(* IEC 61131-3 sources: SJ_AGV/PLC/Standard_functions.4.4.0/Common, 6 files *)

(* ---- DEBUG_FB.ST ---- *)
FUNCTION_BLOCK DEBUG_FB
VAR_EXTERNAL

END_VAR

VAR_INPUT

END_VAR

VAR_OUTPUT

END_VAR

VAR

END_VAR
if debug then
	a:= TRACE_bool('ExecDrvCmd',NDC8.Automatic.ExecDriveCommand);
	a:= TRACE_bool('CancOp',NDC8.LoadOperation.CancelOperation);
	a:= TRACE_dint('TrvlDir',NDC8.VehicleControl.TravelDir);
	a:= TRACE_BOOL('Loaded', input.LoadOnBoard);
	a:= TRACE_DINT('Segm', NDC8.LayoutPosition.Segment);
	a:= TRACE_BOOL('OnLastseg', NDC8.LoadDocking.OnLastSegment);
	a:= TRACE_DINT('StopWord', NDC8.UserDefined.StopWord);
	a:= TRACE_DINT('OpCode', NDC8.LoadOperation.OperationCode);
	a:= TRACE_DINT('OpPar1', NDC8.LoadOperation.OperationParam1);

	debug := false;

end_if;

END_FUNCTION_BLOCK

(* ---- INDICATORS_FB.ST ---- *)
FUNCTION_BLOCK INDICATORS_FB
VAR_EXTERNAL
	(** IN **)
	NDC8 : NDC8_T;
	INPUT : INPUT_T;
	Output : OUTPUT_T;

END_VAR

VAR_INPUT
	SetHeight						: dint;
	ForkTarget,
	AutoInsertNotInsideTargetSafety,
	AutoinsertInProgress,
	SensorsBuzzerTest,
	StartDelayStartWarning,
	LS2000SlowDown					: bool;

END_VAR

VAR_OUTPUT

END_VAR

VAR
	FlashError,
	FlashWarning,
	FlashRight,
	FlashLeft,
	FlashForward,
	FlashBackward,
	FlashSegment : Bool;
	FlashBrakeRel : BOOL;
	ModeAutoTON :TON;

	Display : bool;
	SlowBeep : bool;

END_VAR
(*
------------------------------------------------------------------------------------
 INDICATORS_FB
 ------------------

 Description:
 This PLC controls the flashing of the lights and the sounding of the buzzer.
 The lights and buzzer functionality is made according to safety regulations EN-1525.

-------------------------------------------------------------------------------------*)

(* make default *)
Output.PositionKnownLamp 	:= false;
Output.EmergencyStopLamp 	:= false;
Output.LoadOnBoardLamp	 	:= false;
Output.InSystemLamp			:= false;
Output.FrontLeftLamp 		:= false;
Output.FrontRightLamp 		:= false;
Output.RearLeftLamp 		:= false;
Output.RearRightLamp 		:= false;
Output.WarningBuzzerTop		:= false;
Output.WarningLightTop		:= false;
Output.Buzzer 				:= false;
Output.OPTBuzzer			:= false;

(***************************************************************************************
	Evaluate which signals to set
****************************************************************************************)
(*Emergency stop or any stop flags*)
FlashError	:=	NDC8.VehicleControl.Estop
				or StopRear
				or StopSide
				or StopObstacle
				or StopLift
				or StopLoadChange
				or StopReset
				or StopSteerSync
				or StopForkFarTooHigh
				or StopForkTooHigh
				or StopForkTooLow
				or NDC8.Opt.VehicleStatusID = 11;

FlashBrakeRel := INPUT.Auto = TRUE and NDC8.SDIO.DigitalInput5_BTN_BRK = TRUE;

(*Segment trigger flash*)
FlashSegment := NDC8.VehicleControl.Moving;

(*Segment trigger or Vehical right turn*)
FlashRight 	:= 	Input.SD_Right or Input.DD_Right;

(*Segment trigger or Vehical right turn*)
FlashLeft 	:=	Input.SD_Left or Input.DD_Left;

(*Segment trigger or Vehical Forward*)
FlashForward := Input.SD_Forward;

(*Segment trigger or Vehical Backward*)
FlashBackward := Input.SD_Backward;

(* Special case for when we want to flash both right _and_left *)
(*If FlashRight and FlashLeft then
	  FlashRight	:= NDC8.TurnSignal.RightTurnDistance < NDC8.TurnSignal.LeftTurnDistance;
	  FlashLeft		:= NDC8.TurnSignal.LeftTurnDistance < NDC8.TurnSignal.RightTurnDistance;
End_if;*)

(*Vehicle moving backwards, forks are moving or before starting to drive *)
FlashWarning := (SetHeight > 0 and not ForkTarget )
				or (NDC8.VehicleControl.Moving and NDC8.VehicleControl.TravelDir = 0)
				or INPUT.SafetyScannerSlowDown
				or StartDelayStartWarning
				or (NDC8.Guidance.StopReason = 1
  					and NDC8.Guidance.DistanceToStop < 1500
  					and NDC8.VehicleControl.TravelDir = 1);		(* Vehicle will stop and change travel directions and reverse. *)

(***************************************************************************************)
(*			LAMPS 					*)
(***************************************************************************************)
(* GREEN lamp;	Position known *)
if 	NDC8.Position.Valid then
	if NDC8.VehicleControl.OperationMode = 0 then
		Output.PositionKnownLamp := true;										(* Automatic mode: 		ON 		*)
	else
	 	Output.PositionKnownLamp := Timer.Info;								(* Semi/manual mode: 	BLINK 	*)
	end_if;
end_if;

(***************************************************************************************)
(* WHITE lamp; reset button *)

Output.ResetButtonLamp	:= (StopReset or												(* need reset	*)
					   		StopManual or
					   		AutoInsertNotInsideTargetSafety 								(* vehicle need assistance during autoinsert *)
							)
							and Timer.Info;

(***************************************************************************************)
(* YELLOW lamp; Load on board*)
Output.LoadOnBoardLamp := INPUT.LoadOnBoard and Timer.Info;

(***************************************************************************************)
(* RED lamp; S100 stop *)
Output.EmergencyStopLamp := NDC8.VehicleControl.OperationMode = 0 and StopObstacle and Timer.Error;								(* S100 stop *)

(***************************************************************************************)
(* BLUE lamp; In system *)

if NDC8.VehicleControl.OperationMode = 0 then
	Output.InSystemLamp :=	NDC8.LayoutPosition.InSystem 							(* in system *)
				or (AutoinsertInProgress and NDC8.VehicleControl.Moving and Timer.Warning)

				or (INPUT.Reset_PB  								(*	 on when pressed and outside safety	*)
					and AutoInsertNotInsideTargetSafety
					)
				or (AutoinsertInProgress				(* 	 need more RESET help 	*)
					and not NDC8.VehicleControl.Moving
					and Timer.Info);
end_if;

(***************************************************************************************)
(* SIDE ORANGE lamp; warning/turn indicators *)
InStatus := NDC8.VehicleControl.OperationMode = 0;
ModeAutoTON(IN:=InStatus,PT:=t#2s);	(* Wait 2 sec before flashing when entering auto*)
if TRUE then
	if FlashError then
		Output.RearLeftLamp 	:= Timer.Error;
		Output.RearRightLamp	:= Timer.Error;
		Output.FrontLeftLamp 	:= Timer.Error;
		Output.FrontRightLamp	:= Timer.Error;
		(* vehicle moving or vehicle error both flash *)
		(*
	elsif FlashWarning or FlashSegment then
		Output.RearLeftLamp 	:= Timer.Warning;
		Output.RearRightLamp	:= Timer.Warning;
		Output.FrontLeftLamp 	:= Timer.Warning;
		Output.FrontRightLamp	:= Timer.Warning;*)
	elsif FlashBrakeRel then
		Output.FrontLeftLamp 	:= TRUE;
		Output.RearLeftLamp 	:= TRUE;
		Output.FrontRightLamp 	:= TRUE;
		Output.RearRightLamp 	:= TRUE;
	elsif FlashForward then								(* vehicle turning to the left *)
		Output.FrontLeftLamp 	:= Timer.Warning;
		Output.RearLeftLamp 	:= Timer.Warning;
		Output.FrontRightLamp 	:= Timer.Warning;
		Output.RearRightLamp 	:= Timer.Warning;
	elsif FlashBackward then								(* vehicle turning to the left *)
		Output.FrontLeftLamp 	:= Timer.Warning;
		Output.RearLeftLamp 	:= Timer.Warning;
		Output.FrontRightLamp 	:= Timer.Warning;
		Output.RearRightLamp 	:= Timer.Warning;
	elsif FlashRight then								(* vehicle turning to the right *)
		Output.FrontLeftLamp 	:= false;
		Output.RearLeftLamp 	:= false;
		Output.FrontRightLamp 	:= Timer.Warning;
		Output.RearRightLamp 	:= Timer.Warning;
	elsif FlashLeft then								(* vehicle turning to the left *)
		Output.FrontLeftLamp 	:= Timer.Warning;
		Output.RearLeftLamp 	:= Timer.Warning;
		Output.FrontRightLamp 	:= false;
		Output.RearRightLamp 	:= false;
	elsif NDC8.VehicleControl.Moving = FALSE then
		Output.FrontLeftLamp 	:= TRUE;
		Output.RearLeftLamp 	:= TRUE;
		Output.FrontRightLamp 	:= TRUE;
		Output.RearRightLamp 	:= TRUE;
	end_if;
elsif StopReset then									(* Reset required *)
		Output.FrontLeftLamp 	:= Timer.Info and Timer.Error and Timer.Warning;
		Output.FrontRightLamp 	:= Timer.Info and Timer.Error and Timer.Warning;
		Output.RearLeftLamp 	:= Timer.Info and Timer.Error and Timer.Warning;
		Output.RearRightLamp 	:= Timer.Info and Timer.Error and Timer.Warning;
end_if;

if StopLS2000 or LS2000SlowDown then							(* Vehicle is about to drive into something and hit LS2000! *)
		Output.RearLeftLamp 	:= Timer.Warning;
		Output.RearRightLamp	:= Timer.Warning;
		Output.FrontLeftLamp 	:= Timer.Warning;
		Output.FrontRightLamp	:= Timer.Warning;
end_if;

(***************************************************************************************)
(* 					BUZZERS 					*)
(***************************************************************************************)
(* High frequency tone. Sound only when there is a drive command. *)
InStatus := NDC8.VehicleControl.OperationMode = 0;
ModeAutoTON(IN:=InStatus,PT:=t#3s);	(* Wait 3 sec before buzzing when entering auto *)
Output.Buzzer	:=	(ModeAutoTON.Q and
						NDC8.Automatic.ExecDriveCommand	and
							(FlashError and Timer.Error)				(* Error *)
						 	or
						 	(FlashWarning and Timer.Warning)					(* Info *)
						)
					or SensorsBuzzerTest
					or (StopLS2000 or LS2000SlowDown and Timer.Warning);			(* Vehicle is about to drive into something and hit LS2000! *)

(* OPT 100 BUZZER Low frequency tone *)
OUTPUT.OPTBuzzer	:= StartDelayStartWarning					(* Sound during start or if reset is required. *)
						or
							(StopReset or StopLS2000 or LS2000SlowDown)
							and Timer.Info
							and Timer.Error
							and Timer.Warning
							and SlowBeep;

END_FUNCTION_BLOCK

(* ---- MODECONTROL_FB.ST ---- *)
FUNCTION_BLOCK MODECONTROL_FB
VAR_EXTERNAL
	NDC8 : NDC8_T;
	INPUT : INPUT_T;
	TRUCK : TRUCK_T;

END_VAR

VAR_INPUT

END_VAR

VAR_OUTPUT
		Auto			: bool; (* 8 *)
		Manual			: bool; (* 1 *)
		Semi			: bool; (* 2 *)
		PPA				: bool; (* 4 *)

END_VAR

VAR
	State			: dint;
	SteerModeRT		: r_trig;
	SteerModeRT2	: r_trig;
	SteerMode	: dint;

	StepDelay : TON;

	NoMcdTimer : TON;

END_VAR
(*****************************************************************************************)
(* Truck Modes of Operation:

	Auto  					- full AGV control
	Manual					- Vehicle driven from tiller arm or MCD.
	PPA Tune  				- AGV drive mode, but vehicle controller set to manual mode to allow PPA Tuning

	NDC8.Manual.PlcSelectMask	DINT 	Individually select mask:
		Bit0:PlcAngle 				2#00000
		Bit1:PlcSpeed 				2#00010
		Bit2:PlcSetOperationMode 	2#00100
		Bit3:Reserved 				2#01000
		Bit4:PlcSteerMethod			2#10000
	*)

NDC8.Manual.PlcSelect := true;							(* By default, allow overrides.*)
NDC8.Manual.PlcSelectMask := 0;							(* By default, don't override anything*)

(* only one mode is allowed at one time *)
Auto 			:= word_to_bool(dint_to_word(State) and 16#8);
Manual			:= word_to_bool(dint_to_word(State) and 16#1);
Semi			:= word_to_bool(dint_to_word(State) and 16#2);
PPA 			:= word_to_bool(dint_to_word(State) and 16#4);

INPUT.Auto := Auto;
INPUT.Manual := Manual;
INPUT.Semi := Semi;
INPUT.PPA := PPA;

if NDC8.Mcd.Valid = TRUE and g_StartFindSync = FALSE then

	SteerModeRT(CLK:=Input.ChangeSteerMode_PB);		(* New steer mode requested (Quad vehicle)
															0: 2*SD Anti-parallel
															1: 2*SD Parallel
															2: DiffDrive  				*)
	SteerModeRT2(CLK:=Input.ChangeSteerMode_PB2);

	case State of
	(*****************************************************************************************
				Automatic mode
	*****************************************************************************************)
	0: State := 8;

	8:	NDC8.Manual.PlcSetOperationMode := 0;			(* Operation mode Auto *)
		NDC8.Manual.PlcSelectMask		:= 2#00110;	(* Override Set speed, to allow autinsert from outside safety zone
														 Speed is set in AutoInsert FB. *)

		(**** Exit this mode? ***)
		if NDC8.Mcd.Button2 and NDC8.Mcd.Valid then		(* MCD semi mode *)
			State := 2;

		elsif (NDC8.Mcd.Button3 and NDC8.Mcd.Valid)		(* MCD manual mode *)
			or INPUT.TillerArmDown 						(* Manual arm down, switch to manual mode		*)
			or INPUT.GateOpen
			or INPUT.PlatformNotUpperPos then
				State := 1;

		elsif NDC8.Userdefined.PPAEnable = 2 then		(* Change to PPA mode if set in OPT	expert menu.*)
				State := 4;
		end_if;

	(*****************************************************************************************
				Semi mode (MCD throttle, automatic steering)
	*****************************************************************************************)
	2:	NDC8.Manual.PlcSetOperationMode := 2;			(* Set semi mode *)
		NDC8.Manual.PlcSelectMask 		:= 2#10010;	(* Override operation mode and steer mode (quad) *)

		(**** Exit this mode? ***)
		if NDC8.Mcd.Button1 or not NDC8.Mcd.Valid then		(* If disconnect the MCD or switch modes, to auto *)
			State := 8;

		elsif (NDC8.Mcd.Button3 and NDC8.Mcd.Valid) then	(* If disconnect the MCD or switch modes, to auto *)
			State := 1;
		end_if;

	(*****************************************************************************************
				Manual driving
	*****************************************************************************************)
	1:	NDC8.Manual.PlcSetOperationMode := 1;				(* Set Manual mode 							*)
		StopLoadOP := False;								(* Clear load op cancel stop bit			*)

		if SteerModeRT.q then
			SteerMode:= SteerMode + 1;          			(* Toggle steermode *)
	        if SteerMode > 2 then                  			(* Limit *)
	        	SteerMode:= 0;                				(* Reset *)
			end_if;
	        NDC8.Manual.PLCSteerMode:= SteerMode;   		(* Use steermode *)
		end_if;

		if SteerModeRT2.q then
			SteerMode:= SteerMode - 1;          		(* Toggle steermode *)
	        if SteerMode < 0 then                  		(* Limit *)
	        	SteerMode:= 2;                			(* Reset *)
			end_if;
	        NDC8.Manual.PLCSteerMode:= SteerMode;   	(* Use steermode *)
		end_if;

		if NDC8.Mcd.Valid then								(* If mcd connected						 	*)
			if Input.ZeroSteerAngle_PB then					(* If "set zero angle" key					*)
				NDC8.Manual.PLCAngle 			:= 0;		(* Set angle to 0							*)

				if StopWord = 0 and StopWord2 = 0  then
					NDC8.Manual.PlcSpeed			:= NDC8.Mcd.Speed;
				elsif NDC8.Mcd.Button8 = FALSE then
					NDC8.Manual.PlcSpeed			:= 0;
				elsif NDC8.Mcd.Button8 = TRUE then
					NDC8.Manual.PlcSpeed			:= NDC8.Mcd.Speed;
				end_if;

				NDC8.Manual.PlcSelectMask 		:= 2#10111;(* Override operation mode, steer mode and set angle	*)
			else
				NDC8.Manual.PLCAngle 			:= NDC8.Mcd.Angle / 3;

				if StopWord = 0 and StopWord2 = 0  then
					NDC8.Manual.PlcSpeed			:= NDC8.Mcd.Speed;
				elsif NDC8.Mcd.Button8 = FALSE then
					NDC8.Manual.PlcSpeed			:= 0;
				elsif NDC8.Mcd.Button8 = TRUE then
					NDC8.Manual.PlcSpeed			:= NDC8.Mcd.Speed;
				end_if;

				NDC8.Manual.PlcSelectMask 		:= 2#10111;(* Override operation mode and steer mode		*)
			end_if;
			DisplayStopString(INStatus:=Input.ZeroSteerAngle_PB, StopString:=184, StopValue:=0);
			StopManual := false;

		else
			NDC8.Manual.PlcSelectMask 		:= 2#10101;			(* Override operation mode, set angle and steer mode		*)
			NDC8.Manual.PlcAngle := Input.SteerEncAngle;		(* Follow encoder angle, to start autoinsert with this set angle. *)

			StopManual	:= not Input.GateOpen 					(* Set stop bit while waiting to go to auto.	*)
						and not Input.TillerArmDown
						and not Input.PlatformNotUpperPos
						and not Input.Reset_PB;
			StopReset	:= StopReset OR StopManual; 			(* This stop signal needs to be reset			*)
		end_if;

		(**** Exit this mode? ***)
		if NDC8.Mcd.Valid then									(* If MCD is connected							*)
			if NDC8.Mcd.Button1 then							(* Auto mode on MCD? Switch to automatic mode.	*)
				State := 8;
			elsif NDC8.Mcd.Button2 then							(* Semi mode on mcd? Switch to semi mode		*)
				State := 2;
			end_if;
		else
			if 	not Input.TillerArmDown							(* Tiller arm up								*)
				and not Input.GateOpen							(* and gate closed 								*)
				and not Input.PlatformNotUpperPos				(* and platform up 								*)
				and Input.Reset_PB then							(* and reset push button! 						*)
					State := 8;							(* Switch to automatic mode						*)
			end_if;
		end_if;

	(*****************************************************************************************
				Physical Parameter Adjust (PPA)
	*****************************************************************************************)

	4:	NDC8.Manual.PlcSetOperationMode  := 1;			(* Set Manual mode								*)
		NDC8.Manual.PlcSelectMask 		 := 2#00100;	(* Override operation mode 						*)

		(**** Exit this mode? ***)
		if INPUT.TillerArmDown
			or INPUT.GateOpen
			or INPUT.PlatformNotUpperPos then
				State := 1;						(* Manual arm down, switch to manual mode		*)

		elsif NDC8.Userdefined.PPAEnable <> 2 then		(* PPA symbol changed? Go back to auto.			*)
				State := 8;
		end_if;

	end_case;

	NoMcdTimer(IN:= FALSE);
elsif NDC8.Mcd.Valid = FALSE and g_StartFindSync = FALSE and g_ErrorCode = 0 then

	NoMcdTimer(IN:= TRUE, PT:=t#5s);

;
end_if;

(**************************************************************************************)
(* Update Display *)

DisplayStopString(INStatus:=StopManual, StopString:=85, StopValue:=0);

END_FUNCTION_BLOCK

(* ---- STOPWORD_FB.ST ---- *)
FUNCTION_BLOCK STOPWORD_FB
VAR_EXTERNAL
	NDC8 : NDC8_T;
END_VAR

VAR_INPUT
END_VAR

VAR_OUTPUT
END_VAR

VAR
	WaitingForSteerWheelTurn : bool;
	Stop_RT : R_Trig;
	Stop_FT : F_Trig;
	TempValue : dint ;
	StopTON : ton;
END_VAR
(**************************************************************************************)
(* LOAD OPERATION STOP *)
(* Do not enter station w/o OP code *)
(*StopNoOPCode := NDC8.LoadOperation.OperationCode = 0
				and NDC8.Automatic.ExecDriveCommand;
DisplayStopString(InStatus:=StopNoOPCode, StopString:=94, StopValue:=0);

*)

(**************************************************************************************)
(* Waiting for steering wheel to turn *)
(* If no other errors, it's most likely the steer wheel which is not within NDC8.Vehicle.WaitForWheelTurnMaxAngle. *)

WaitingForSteerWheelTurn := NDC8.Automatic.ExecDriveCommand
							and NDC8.CanOpenMaster.NMTState = 5
							and NDC8.CanOpenMaster.State = 0
							and NDC8.Position.Valid
							and not NDC8.Vehicle.Blocked
							and not NDC8.VehicleControl.QuickStop
							and not NDC8.VehicleControl.Stop
							and not NDC8.VehicleControl.EStop
							and not NDC8.VehicleControl.SensorStopEnable
							and NDC8.VehicleControl.SetSpeed = 0
							and abs(Input.SteerEncAngle - Output.SetValueSteer) > NDC8.Vehicle.WaitForWheelTurnMaxAngle;

DisplayStopString(InStatus:=WaitingForSteerWheelTurn, StopString:=138, StopValue:=0);

StopSteerSync	:= not INPUT.SteerEncSyncValid;
DisplayStopString(InStatus:=StopSteerSync, StopString:=181, StopValue:=0);

DisplayStopString(InStatus:=StopByOM_PLC, StopString:=200, StopValue:=0);
DisplayStopString(InStatus:=StopByErrorCode, StopString:=201, StopValue:=0);
DisplayStopString(InStatus:=StopBatLowOT, StopString:=202, StopValue:=0);
DisplayStopString(InStatus:=StopFindSync, StopString:=203, StopValue:=0);
DisplayStopString(InStatus:=StopRobotNotIdle, StopString:=204, StopValue:=0);
DisplayStopString(InStatus:=StopByBCD, StopString:=205, StopValue:=0);

DisplayStopString(InStatus:=StopLift, 				StopString:=210, StopValue:=0);
DisplayStopString(InStatus:=StopRear,				StopString:=211, StopValue:=0);
DisplayStopString(InStatus:=StopSafety, 			StopString:=212, StopValue:=0);
DisplayStopString(InStatus:=StopFailureCAN, 		StopString:=213, StopValue:=0);
DisplayStopString(InStatus:=StopStartDelay,	 		StopString:=214, StopValue:=0);
DisplayStopString(InStatus:=StopFlex, 				StopString:=215, StopValue:=0);
DisplayStopString(InStatus:=StopSoft, 				StopString:=216, StopValue:=0);
DisplayStopString(InStatus:=StopLoadChange,	 		StopString:=217, StopValue:=0);
DisplayStopString(InStatus:=StopObstacle, 			StopString:=218, StopValue:=0);
DisplayStopString(InStatus:=StopEStopChainError, 	StopString:=219, StopValue:=0);
DisplayStopString(InStatus:=StopSteerSync, 			StopString:=220, StopValue:=0);
DisplayStopString(InStatus:=StopEstopButton, 		StopString:=221, StopValue:=0);
DisplayStopString(InStatus:=StopSide, 				StopString:=222, StopValue:=0);
DisplayStopString(InStatus:=StopReset,				StopString:=223, StopValue:=0);
DisplayStopString(InStatus:=StopNoOpCode, 			StopString:=224, StopValue:=0);
DisplayStopString(InStatus:=StopManual, 			StopString:=225, StopValue:=0);
DisplayStopString(InStatus:=StopCharge, 			StopString:=226, StopValue:=0);
DisplayStopString(InStatus:=StopClamp, 				StopString:=227, StopValue:=0);
DisplayStopString(InStatus:=StopFailCode, 			StopString:=228, StopValue:=0);
DisplayStopString(InStatus:=StopResetButton, 		StopString:=229, StopValue:=0);
DisplayStopString(InStatus:=StopLoadOP, 			StopString:=230, StopValue:=0);
DisplayStopString(InStatus:=StopBumperFault, 		StopString:=231, StopValue:=0);
DisplayStopString(InStatus:=StopObstacleFault, 		StopString:=232, StopValue:=0);
DisplayStopString(InStatus:=StopTruckDriveSafeState,StopString:=233, StopValue:=0);
DisplayStopString(InStatus:=StopLS2000, 			StopString:=234, StopValue:=0);
DisplayStopString(InStatus:=StopHalt, 				StopString:=235, StopValue:=0);
DisplayStopString(InStatus:=StopLoadDroppedWhileUnloading, StopString:=236, StopValue:=0);
DisplayStopString(InStatus:=StopSpinningWheel, 		StopString:=237, StopValue:=0);
DisplayStopString(InStatus:=StopForkTooLow, 		StopString:=238, StopValue:=0);
DisplayStopString(InStatus:=StopForkTooHigh, 		StopString:=239, StopValue:=0);
DisplayStopString(InStatus:=StopForkFarTooHigh, 	StopString:=240, StopValue:=0);
DisplayStopString(InStatus:=StopChargeStationMissing, StopString:=241, StopValue:=0);

DisplayStopString(InStatus:=StopByCanErr_Node1, StopString:=244, StopValue:=0);
DisplayStopString(InStatus:=StopByCanErr_Node2, StopString:=245, StopValue:=0);
DisplayStopString(InStatus:=StopByCanErr_Node3, StopString:=246, StopValue:=0);
DisplayStopString(InStatus:=StopByCanErr_Node4, StopString:=247, StopValue:=0);
DisplayStopString(InStatus:=StopByCanErr_Node5, StopString:=248, StopValue:=0);
DisplayStopString(InStatus:=StopByCanErr_Node6, StopString:=249, StopValue:=0);
DisplayStopString(InStatus:=StopByCanErr_Node7, StopString:=250, StopValue:=0);
DisplayStopString(InStatus:=StopByCanErr_Node8, StopString:=251, StopValue:=0);
DisplayStopString(InStatus:=StopByCanErr_Node9, StopString:=252, StopValue:=0);
DisplayStopString(InStatus:=StopByCanErr_Node10, StopString:=253, StopValue:=0);

(**************************************************************************************)
(* QUICK STOP  (Stop with emergency deceleration ramp) 								  *)
(*NDC8.VehicleControl.QuickStop := StopFlex or StopObstacle or StopSafety;
*)
DisplayStopString(INStatus:=NDC8.VehicleControl.QuickStop, StopString:=179, StopValue:=0);

(**************************************************************************************)
(* STOP WORD sets stop signal 														  *)
NDC8.VehicleControl.Stop 	:= 	(Input.Auto and (DWORD_TO_BOOL(StopWord) or DWORD_TO_BOOL(StopWord2))) or
								(Input.Manual and NDC8.Mcd.Button8 = FALSE and (DWORD_TO_BOOL(StopWord) or DWORD_TO_BOOL(StopWord2)));
NDC8.UserDefined.StopWord	:=	DWORD_TO_DINT(StopWord);
NDC8.OMPLC.StopWord			:=	DWORD_TO_INT(StopWord);

StopTON(IN:=NDC8.VehicleControl.Stop,PT:=t#10s);
Stop_RT(CLK:=StopTON.q);
if Stop_RT.Q and not StopStartDelay then
	TempValue:=DWord_To_DINT(StopWord);
end_if;

(* Send event that stopword has been cleared. * )
Stop_FT(CLK:=NDC8.VehicleControl.Stop);
if Stop_FT.q then
	EventQueue(EventCode:=101,Par1:=NDC8.Vehicle.VehicleID,Par2:=0,Par3:=0,Par4:=0);
end_if;
*)

END_FUNCTION_BLOCK

(* ---- Timer_FB.ST ---- *)
FUNCTION_BLOCK Timer_FB
VAR_OUTPUT
	Error : bool;
	Warning : bool;
	Info : bool;
	Display : bool;
	SlowBeep : bool;

END_VAR

VAR
	TimerError 		: blink;
	TimerWarning 	: blink;
	TimerInfo 		: blink;
	TimerDisplay	: blink;
	TimerSlowBeep	: blink;
END_VAR
(*
------------------------------------------------------------------------------------
 FREERUN
 -------

 Description:
 Creates different outputs that will look like a freerunning timer.
 Outputs will toggle with different timebase.
 They are all defined globally.
------------------------------------------------------------------------------------   *)

TimerError	(CYCLE :=t#240ms,RUN:=true);
TimerWarning(CYCLE :=t#480ms,RUN:=true);
TimerInfo	(CYCLE :=t#960ms,RUN:=true);
TimerDisplay(CYCLE :=t#2s,RUN:=true);
TimerSlowBeep(CYCLE :=t#5s,RUN:=true);

Error		:= TimerError.Q1;
Warning	:= TimerWarning.Q1;
Info		:= TimerInfo.Q1;
Display	:= TimerDisplay.Q1;
SlowBeep	:= TimerSlowBeep.Q1;

END_FUNCTION_BLOCK

(* ---- TX_STATUS_FB.ST ---- *)
FUNCTION_BLOCK TX_STATUS_FB
VAR_EXTERNAL
	NDC8 : NDC8_T;
	Input : Input_T;

END_VAR

VAR_INPUT

END_VAR

VAR_OUTPUT

END_VAR

VAR

	Load_F : F_Trig;
	Load_F_FLAG : BOOL;

	Load_F_Timer : TON;

	BCD_Compare_R : F_Trig;
	BCD_Fail_R : F_Trig;

	BatLowR : R_Trig;
	BatLowF : F_Trig;

	ErrorCodeD : DINT;
	LastErrorCode : Word := 0;
	ErrorTrigFlag : bool;
	ErrorTrigR : R_Trig;
	ErrorTrigF : F_Trig;

	InsertDone : BOOL;
	InsertDoneR : R_Trig;

	PowerOffR	: R_Trig;

	WaitChargeR	: R_Trig;
	WaitChargeF	: F_Trig;

	ChargingR : R_Trig;
	ChargingF : F_Trig;

	ChargeDoneR : R_Trig;

	LoadStatusR :R_Trig;
	LoadStatusF :F_Trig;

	ManualModeR :R_Trig;
	ManualModeF :F_Trig;

	LostR :R_Trig;
	LostF :F_Trig;

	LocalModeR :R_Trig;
	LocalModeF :F_Trig;

	LocalInterlockFailCodeD : DINT;
	LocalInterlockFailFlag : bool;
	LocalInterlockFailR :R_Trig;

	DriveOutR : R_Trig;

	BrakeReleaseR : R_Trig;
	BrakeReleaseF : F_Trig;

	BeamStop_R : R_Trig;
	BeamStop_F : F_Trig;

	BlockFlagR : R_Trig;
	BlockFlagF : F_Trig;
	BlockModeFlag : BOOL;

	BCDReadFailR :R_Trig;

	(* Battery *)
	ChrgFlag_R_L : BOOL;
	TX_LowBatt_R : R_Trig;
	TX_ChgComp_R : R_Trig;
	Chrg_Right_Left_R : R_Trig;
	TX_Load_R : R_Trig;

	DINT_BMS2 : DINT;
	DINT_BMS3 : DINT;
	DINT_BMS_BatV : DINT;
	DINT_BMS_BatT : DINT;
	DINT_BMS_BatC : DINT;
	DINT_BMS_BatA : DINT;
	DINT_BMS_Main : DINT;
	DINT_BMS_Chan : DINT;
	DINT_BMS_ID4L : DINT;
	DINT_BMS_ID4H : DINT;

END_VAR
(*
------------------------------------------------------------------------------------
 TX_status
 ------------------

 Description:
 Sends status bits to master controller.

-------------------------------------------------------------------------------------*)
(*TxStatus bits*)

OM_PLC_Word1 := INT_TO_WORD(NDC8.OMPLC.ChargeOM);
OM_PLC_Word2 := INT_TO_WORD(NDC8.OMPLC.Stop_OM);

NDC8.PLC_Application.TxStatusBit0_Load := INPUT.LoadOnBoard;
NDC8.PLC_Application.TxStatusBit1_EaLD := PLC_RX01_Bit_EnableLD_i;

if NDC8.LoadOperation.OperationCode <> 0 then
	NDC8.PLC_Application.TxStatusBit2_HaveCmd := true;	(*Operation Code OK*)
else
	NDC8.PLC_Application.TxStatusBit2_HaveCmd := false;	(*Operation Code OK*)
end_if;

NDC8.PLC_Application.TxStatusBit3_RelBRK := NDC8.SDIO.DigitalInput5_BTN_BRK; (*Brake release*)

Load_F(CLK:=PLC_RX01_Bit_Load_i);

if Load_F.Q then
	Load_F_FLAG := TRUE;
end_if;

Load_F_Timer(IN:=Load_F_FLAG, PT:=t#1s);

if Load_F_Timer.Q then
	Load_F_FLAG := FALSE;
end_if;

if (OM_PLC_W1_Bit_WaitCharge = TRUE and OM_PLC_W1_Bit_SetLowBatt = FALSE) or OM_PLC_W1_Bit_WaitOrder = TRUE then

	if NDC8.PLC_Application.TxStatusBit5_WaitLow = FALSE then
		NDC8.PLC_Application.TxStatusBit5_WaitLow := TRUE; (*Charge Wait*)
	elsif Load_F_FLAG = TRUE then
		OM_PLC_W1_Bit_WaitCharge := FALSE;
		NDC8.PLC_Application.TxStatusBit5_WaitLow := FALSE;
		Load_F_FLAG := FALSE;
	end_if;

else
	NDC8.PLC_Application.TxStatusBit5_WaitLow := FALSE; (*Charge Wait*)
end_if;

NDC8.PLC_Application.TxStatusBit4_LowBatt := (INPUT.LowBattery or NDC8.Userdefined.LowBatSim or OM_PLC_W1_Bit_SetLowBatt)and NDC8.PLC_Application.TxStatusBit5_WaitLow = FALSE ; (*Battery Low*)

NDC8.PLC_Application.TxStatusBit6_Charge := NDC8.SDIO.DigitalOutput16_RIGHTMGS OR NDC8.SDIO.DigitalOutput12_LEFTMGS; (*Charging*)

(*
if PLC_RX03_Bit_STw_FullCg = TRUE or PLC_RX15_Bit_BMS_ChgCmp = TRUE then
	NDC8.PLC_Application.TxStatusBit7_ChgComp := TRUE;
elsif PLC_RX01_Bit_ChrgIdle = TRUE or NDC8.PLC_Application.TxStatusBit9_EStop = TRUE then
	NDC8.PLC_Application.TxStatusBit7_ChgComp := FALSE;
end_if;
*)

NDC8.PLC_Application.TxStatusBit8_Manual := PLC_TX01_Bit_ManMode; (*Manual Mode*)
NDC8.PLC_Application.TxStatusBit9_EStop := NDC8.VehicleControl.Estop or StopEstopButton; (*Emergency Stop*)
NDC8.PLC_Application.TxStatusBit10_Blocked := PLC_TX03_Bit_STr_Block;  (*Blocked*)
NDC8.PLC_Application.TxStatusBit11_IrStop := false; (*Obstacle sensor Stop*)
NDC8.PLC_Application.TxStatusBit12_LostP := g_ErrorCode = 137; (*Lost Position*)
NDC8.PLC_Application.TxStatusBit13 := false;
NDC8.PLC_Application.TxStatusBit14 := false;
NDC8.PLC_Application.TxStatusBit15 := false;

(*Tx Event*)
(*---------------------------------------------------------------------------*)

(* User Event 3: Battery ON *)
BatLowR(CLK:= NDC8.PLC_Application.TxStatusBit4_LowBatt);
if BatLowR.Q and NDC8.Master.MasterLinkUp then
	EventQueue(EventCode:=3,
		Par1:=NDC8.LayoutPosition.Segment,
		Par2:=0,
		Par3:=0,
		Par4:=0);
a:=TRACE_DINT('EventCode', EventQueue.EventCode);
end_if;

(* User Event 33: Battery OFF *)
BatLowF(CLK:= NDC8.PLC_Application.TxStatusBit4_LowBatt);
if BatLowF.Q and NDC8.Master.MasterLinkUp then
	EventQueue(EventCode:=33,
		Par1:=NDC8.LayoutPosition.Segment,
		Par2:=0,
		Par3:=0,
		Par4:=0);
a:=TRACE_DINT('EventCode', EventQueue.EventCode);
end_if;

(* User Event 2: Load Status ON *)
LoadStatusR(CLK:= PLC_RX01_Bit_Load_i);
if LoadStatusR.Q and NDC8.Master.MasterLinkUp then
	EventQueue(EventCode:=2,
		Par1:=NDC8.LayoutPosition.Segment,
		Par2:=0,
		Par3:=0,
		Par4:=0);
a:=TRACE_DINT('EventCode', EventQueue.EventCode);
end_if;

(* User Event 32: Load Status OFF *)
LoadStatusF(CLK:= PLC_RX01_Bit_Load_i);
if LoadStatusF.Q and NDC8.Master.MasterLinkUp then
	EventQueue(EventCode:=32,
		Par1:=NDC8.LayoutPosition.Segment,
		Par2:=0,
		Par3:=0,
		Par4:=0);
a:=TRACE_DINT('EventCode', EventQueue.EventCode);
end_if;

(* User Event 1: Error ON ErrorCode *)
(* User Event 91: Error ON Current Segment*)
(* User Event 92: Error ON Mode 0:Auto 1:Manual*)

if g_ErrorCode = 0 then
	ErrorTrigFlag := FALSE;
	LastErrorCode := 0;
elsif LastErrorCode <> g_ErrorCode then
	ErrorTrigFlag := TRUE;
end_if;

ErrorTrigR(CLK:= ErrorTrigFlag);

if ErrorTrigR.Q and NDC8.Master.MasterLinkUp then

	LastErrorCode := g_ErrorCode;
	ErrorCodeD := WORD_TO_DINT(LastErrorCode);

	EventQueue(EventCode:=1,
			Par1:=ErrorCodeD,
			Par2:=0,
			Par3:=0,
			Par4:=0);
	a:=TRACE_DINT('EventCode', EventQueue.EventCode);

	EventQueue(EventCode:=91,
			Par1:=NDC8.LayoutPosition.Segment,
			Par2:=0,
			Par3:=0,
			Par4:=0);
	a:=TRACE_DINT('EventCode', EventQueue.EventCode);

	if INPUT.Auto then
		EventQueue(EventCode:=92,
			Par1:=0,
			Par2:=0,
			Par3:=0,
			Par4:=0);
		a:=TRACE_DINT('EventCode', EventQueue.EventCode);
	else
		EventQueue(EventCode:=92,
			Par1:=1,
			Par2:=0,
			Par3:=0,
			Par4:=0);
		a:=TRACE_DINT('EventCode', EventQueue.EventCode);
	end_if;

	LastErrorCode := g_ErrorCode;

end_if;

(* User Event 31: Error OFF *)

(*PLC*)
ErrorTrigF(CLK:= ErrorTrigFlag);

if ErrorTrigF.Q and NDC8.Master.MasterLinkUp then

	ErrorCodeD := WORD_TO_DINT(LastErrorCode);
	EventQueue(EventCode:=31,
		Par1:=ErrorCodeD,
		Par2:=0,
		Par3:=0,
		Par4:=0);
	a:=TRACE_DINT('EventCode', EventQueue.EventCode);
end_if;

(* User Event 61: Insert ON *)

InsertDone := NDC8.Autoinsert.StatusID = 5;

InsertDoneR(CLK:= InsertDone);
if InsertDoneR.Q and NDC8.Master.MasterLinkUp then
	EventQueue(EventCode:=61,
		Par1:=NDC8.LayoutPosition.Segment,
		Par2:=0,
		Par3:=0,
		Par4:=0);
	a:=TRACE_DINT('EventCode', EventQueue.EventCode);
end_if;

(* User Event 93: Auto Power OFF *)
PowerOffR(CLK:= g_PowerOffFlag);
if PowerOffR.Q and NDC8.Master.MasterLinkUp then
	EventQueue(EventCode:=93,
		Par1:=NDC8.LayoutPosition.Segment,
		Par2:=0,
		Par3:=0,
		Par4:=0);
	a:=TRACE_DINT('EventCode', EventQueue.EventCode);
end_if;

(* User Event 4: Charge Wait ON *)
WaitChargeR(CLK:= NDC8.PLC_Application.TxStatusBit5_WaitLow);
if WaitChargeR.Q and NDC8.Master.MasterLinkUp then
	EventQueue(EventCode:=4,
		Par1:=NDC8.LayoutPosition.Segment,
		Par2:=0,
		Par3:=0,
		Par4:=0);
	a:=TRACE_DINT('EventCode', EventQueue.EventCode);
end_if;

(* User Event 34: Charge Wait OFF *)
WaitChargeF(CLK:= NDC8.PLC_Application.TxStatusBit5_WaitLow);
if WaitChargeF.Q and NDC8.Master.MasterLinkUp then
	EventQueue(EventCode:=34,
		Par1:=NDC8.LayoutPosition.Segment,
		Par2:=0,
		Par3:=0,
		Par4:=0);
	a:=TRACE_DINT('EventCode', EventQueue.EventCode);
end_if;

(* User Event 6: Charge Complete *)
ChargeDoneR(CLK:= NDC8.PLC_Application.TxStatusBit7_ChgComp);
if ChargeDoneR.Q and NDC8.Master.MasterLinkUp then
	EventQueue(EventCode:=6,
		Par1:=NDC8.LayoutPosition.Segment,
		Par2:=0,
		Par3:=0,
		Par4:=0);
	a:=TRACE_DINT('EventCode', EventQueue.EventCode);
end_if;

(* User Event 5: Charging ON*)
ChargingR(CLK:= NDC8.PLC_Application.TxStatusBit6_Charge);
if ChargingR.Q and NDC8.Master.MasterLinkUp then
	EventQueue(EventCode:=5,
		Par1:=NDC8.LayoutPosition.Segment,
		Par2:=0,
		Par3:=0,
		Par4:=0);
	a:=TRACE_DINT('EventCode', EventQueue.EventCode);
end_if;

(* User Event 35: Charging OFF*)
ChargingF(CLK:= NDC8.PLC_Application.TxStatusBit6_Charge);
if ChargingF.Q and NDC8.Master.MasterLinkUp then
	EventQueue(EventCode:=35,
		Par1:=NDC8.LayoutPosition.Segment,
		Par2:=0,
		Par3:=0,
		Par4:=0);
	a:=TRACE_DINT('EventCode', EventQueue.EventCode);
end_if;

(* User Event 7: Manual Mode ON*)
ManualModeR(CLK:= PLC_TX01_Bit_ManMode);
if ManualModeR.Q and NDC8.Master.MasterLinkUp then
	EventQueue(EventCode:=7,
		Par1:=NDC8.LayoutPosition.Segment,
		Par2:=0,
		Par3:=0,
		Par4:=0);
	a:=TRACE_DINT('EventCode', EventQueue.EventCode);
end_if;

(* User Event 37: Manaul Mode OFF*)
ManualModeF(CLK:= PLC_TX01_Bit_ManMode);
if ManualModeF.Q and NDC8.Master.MasterLinkUp then
	EventQueue(EventCode:=37,
		Par1:=NDC8.LayoutPosition.Segment,
		Par2:=0,
		Par3:=0,
		Par4:=0);
	a:=TRACE_DINT('EventCode', EventQueue.EventCode);
end_if;

(* User Event 10: Lost ON*)
LostF(CLK:= NDC8.LayoutPosition.InSystem);
if LostF.Q and NDC8.Master.MasterLinkUp then
	EventQueue(EventCode:=10,
		Par1:=NDC8.LayoutPosition.Segment,
		Par2:=0,
		Par3:=0,
		Par4:=0);
	a:=TRACE_DINT('EventCode', EventQueue.EventCode);
end_if;

(* User Event 40: Lost OFF*)
LostR(CLK:= NDC8.LayoutPosition.InSystem);
if LostR.Q and NDC8.Master.MasterLinkUp then
	EventQueue(EventCode:=40,
		Par1:=NDC8.LayoutPosition.Segment,
		Par2:=0,
		Par3:=0,
		Par4:=0);
	a:=TRACE_DINT('EventCode', EventQueue.EventCode);
end_if;

(* User Event 11: Local Mode ON*)
LocalModeR(CLK:= PLC_TX01_Bit_LocalMode);
if LocalModeR.Q and NDC8.Master.MasterLinkUp then
	EventQueue(EventCode:=11,
		Par1:=NDC8.LayoutPosition.Segment,
		Par2:=0,
		Par3:=0,
		Par4:=0);
	a:=TRACE_DINT('EventCode', EventQueue.EventCode);
end_if;

(* User Event 41: Local Mode OFF*)
LocalModeF(CLK:= PLC_TX01_Bit_LocalMode);
if LocalModeF.Q and NDC8.Master.MasterLinkUp then
	EventQueue(EventCode:=41,
		Par1:=NDC8.LayoutPosition.Segment,
		Par2:=0,
		Par3:=0,
		Par4:=0);
	a:=TRACE_DINT('EventCode', EventQueue.EventCode);
end_if;

if PLC_TX04_Bit_Cancel_ST = FALSE then
	(* User Event 71: Local Interlock Fail*)
	if PLC_RX_Word10_STw_ILEr <> 0 then
		LocalInterlockFailFlag := TRUE;
	else
		LocalInterlockFailFlag := FALSe;
	end_if;

	LocalInterlockFailR(CLK:= LocalInterlockFailFlag);
	if LocalInterlockFailR.Q and NDC8.Master.MasterLinkUp then

		if PLC_RX_Word10_STw_ILEr = 1 then
			LocalInterlockFailCodeD := 243;
		elsif PLC_RX_Word10_STw_ILEr = 2 then
			LocalInterlockFailCodeD := 242;
		elsif PLC_RX_Word10_STw_ILEr = 3 then
			LocalInterlockFailCodeD := 245;
		elsif PLC_RX_Word10_STw_ILEr = 4 then
			LocalInterlockFailCodeD := 259;
		elsif PLC_RX_Word10_STw_ILEr = 5 then
			LocalInterlockFailCodeD := 260;
		end_if;

		EventQueue(EventCode:=71,
			Par1:=LocalInterlockFailCodeD,
			Par2:=0,
			Par3:=0,
			Par4:=0);
		a:=TRACE_DINT('EventCode', EventQueue.EventCode);
	end_if;
end_if;

(* User Event 72: Drive Out Request*)
DriveOutR(CLK:= PLC_RX04_Bit_STw_DrvOut);

if DriveOutR.Q and NDC8.Master.MasterLinkUp then
	EventQueue(EventCode:=72,
		Par1:=NDC8.LayoutPosition.Segment,
		Par2:=0,
		Par3:=0,
		Par4:=0);
	a:=TRACE_DINT('EventCode', EventQueue.EventCode);
end_if;

(* User Event 12: Brake Release ON *)
BrakeReleaseR(CLK:= NDC8.SDIO.DigitalInput5_BTN_BRK);

if BrakeReleaseR.Q and NDC8.Master.MasterLinkUp then
	EventQueue(EventCode:=12,
		Par1:=NDC8.LayoutPosition.Segment,
		Par2:=0,
		Par3:=0,
		Par4:=0);
	a:=TRACE_DINT('EventCode', EventQueue.EventCode);
end_if;

(* User Event 42: Brake Release OFF *)
BrakeReleaseF(CLK:= NDC8.SDIO.DigitalInput5_BTN_BRK);

if BrakeReleaseF.Q and NDC8.Master.MasterLinkUp then
	EventQueue(EventCode:=42,
		Par1:=NDC8.LayoutPosition.Segment,
		Par2:=0,
		Par3:=0,
		Par4:=0);
	a:=TRACE_DINT('EventCode', EventQueue.EventCode);
end_if;

(* User Event 8: Block ON *)
if NDC8.Automatic.SetOrderMode = 1 or NDC8.Automatic.SetOrderMode = 3 then
	BlockModeFlag := TRUE;
else
	BlockModeFlag := FALSE;
end_if;

BlockFlagR(CLK:=BlockModeFlag);
if BlockFlagR.Q and NDC8.Master.MasterLinkUp then
	EventQueue(EventCode:=8,
		Par1:=NDC8.LayoutPosition.Segment,
		Par2:=0,
		Par3:=0,
		Par4:=0);
	a:=TRACE_DINT('EventCode', EventQueue.EventCode);
end_if;

(* User Event 38: Block OFF *)
BlockFlagF(CLK:=BlockModeFlag);
if BlockFlagF.Q and NDC8.Master.MasterLinkUp then
	EventQueue(EventCode:=38,
		Par1:=NDC8.LayoutPosition.Segment,
		Par2:=0,
		Par3:=0,
		Par4:=0);
	a:=TRACE_DINT('EventCode', EventQueue.EventCode);
end_if;

(* User Event 9: Beam Sensor Stop ON *)
BeamStop_R(CLK:=StopObstacle);
if BeamStop_R.Q and NDC8.Master.MasterLinkUp then
	EventQueue(EventCode:=9,
		Par1:=NDC8.LayoutPosition.Segment,
		Par2:=0,
		Par3:=0,
		Par4:=0);
	a:=TRACE_DINT('EventCode', EventQueue.EventCode);
end_if;

(* User Event 39: Beam Sensor Stop OFF*)
BeamStop_F(CLK:=StopObstacle);
if BeamStop_F.Q and NDC8.Master.MasterLinkUp then
	EventQueue(EventCode:=39,
		Par1:=NDC8.LayoutPosition.Segment,
		Par2:=0,
		Par3:=0,
		Par4:=0);
	a:=TRACE_DINT('EventCode', EventQueue.EventCode);
end_if;

(* User Event 71: BCD Read Fail*)
BCD_Compare_R(CLK:=OM_PLC_W2_Bit_Err_Comp);

if BCD_Compare_R.Q and NDC8.Master.MasterLinkUp then
	EventQueue(EventCode:=71,
		Par1:=155,
		Par2:=0,
		Par3:=0,
		Par4:=0);
	a:=TRACE_DINT('EventCode', EventQueue.EventCode);
end_if;

BCDReadFailR(CLK:=OM_PLC_W2_Bit_Err_BCR);

if BCDReadFailR.Q and NDC8.Master.MasterLinkUp then
	EventQueue(EventCode:=71,
		Par1:=156,
		Par2:=0,
		Par3:=0,
		Par4:=0);
	a:=TRACE_DINT('EventCode', EventQueue.EventCode);
end_if;

(* Bat Event Trig *)
	ChrgFlag_R_L := NDC8.PointTrigger.Bit9_Chrg_Right or NDC8.PointTrigger.Bit10_Chrg_Left;
	TX_LowBatt_R(CLK:= NDC8.PLC_Application.TxStatusBit4_LowBatt);
	TX_ChgComp_R(CLK:= NDC8.PLC_Application.TxStatusBit7_ChgComp);
	Chrg_Right_Left_R(CLK:= ChrgFlag_R_L);
	TX_Load_R(CLK:= NDC8.PLC_Application.TxStatusBit0_Load);

	BMS_EnaEvent := 16#35C;

(* Bat_Low Event *)

	DINT_BMS2 := WORD_TO_DINT(PLC_RX_Word14_BMS_2);
	DINT_BMS3 := WORD_TO_DINT(PLC_RX_Word15_BMS_3);
	DINT_BMS_BatV := WORD_TO_DINT(PLC_RX_Word16_BMS_BatV);
	DINT_BMS_BatT := WORD_TO_DINT(PLC_RX_Word17_BMS_BatT);
	DINT_BMS_BatC := WORD_TO_DINT(PLC_RX_Word18_BMS_BatC);
	DINT_BMS_BatA := WORD_TO_DINT(PLC_RX_Word19_BMS_BatA);
	DINT_BMS_Main := WORD_TO_DINT(PLC_RX_Word21_BMS_Main);
	DINT_BMS_Chan := WORD_TO_DINT(PLC_RX_Word22_BMS_Chan);
	DINT_BMS_ID4L := WORD_TO_DINT(PLC_RX_Word23_BMS_ID4L);
	DINT_BMS_ID4H := WORD_TO_DINT(PLC_RX_Word24_BMS_ID4H);

	if TX_LowBatt_R.Q and EnaBMSEv01 = TRUE then
		(* BMS_ev11 *)
		EventQueue(EventCode:=81,
			Par1:=DINT_BMS2,
			Par2:=0,
			Par3:=0,
			Par4:=0);
		a:=TRACE_DINT('EventCode', EventQueue.EventCode);
	end_if;

	if TX_LowBatt_R.Q and EnaBMSEv02 = TRUE then
		(* BMS_ev12 *)
		EventQueue(EventCode:=82,
			Par1:=DINT_BMS3,
			Par2:=0,
			Par3:=0,
			Par4:=0);
		a:=TRACE_DINT('EventCode', EventQueue.EventCode);
	end_if;

	if TX_LowBatt_R.Q and EnaBMSEv03 = TRUE then
		(* BMS_ev13 *)
		EventQueue(EventCode:=83,
			Par1:=DINT_BMS_BatV,
			Par2:=0,
			Par3:=0,
			Par4:=0);
		a:=TRACE_DINT('EventCode', EventQueue.EventCode);
	end_if;

	if TX_LowBatt_R.Q and EnaBMSEv04 = TRUE then
		(* BMS_ev14 *)
		EventQueue(EventCode:=84,
			Par1:=DINT_BMS_BatT,
			Par2:=0,
			Par3:=0,
			Par4:=0);
		a:=TRACE_DINT('EventCode', EventQueue.EventCode);
	end_if;

	if TX_LowBatt_R.Q and EnaBMSEv05 = TRUE then
		(* BMS_ev15 *)
		EventQueue(EventCode:=85,
			Par1:=DINT_BMS_BatC,
			Par2:=0,
			Par3:=0,
			Par4:=0);
		a:=TRACE_DINT('EventCode', EventQueue.EventCode);
	end_if;

	if TX_LowBatt_R.Q and EnaBMSEv06 = TRUE then
		(* BMS_ev16 *)
		EventQueue(EventCode:=86,
			Par1:=DINT_BMS_BatA,
			Par2:=0,
			Par3:=0,
			Par4:=0);
		a:=TRACE_DINT('EventCode', EventQueue.EventCode);
	end_if;

	if TX_LowBatt_R.Q and EnaBMSEv07 = TRUE then
		(* BMS_ev17 *)
		EventQueue(EventCode:=87,
			Par1:=DINT_BMS_Main,
			Par2:=0,
			Par3:=0,
			Par4:=0);
		a:=TRACE_DINT('EventCode', EventQueue.EventCode);
	end_if;

	if TX_LowBatt_R.Q and EnaBMSEv08 = TRUE then
		(* BMS_ev18 *)
		EventQueue(EventCode:=88,
			Par1:=DINT_BMS_Chan,
			Par2:=0,
			Par3:=0,
			Par4:=0);
		a:=TRACE_DINT('EventCode', EventQueue.EventCode);
	end_if;

(* Chg_Comp Event *)
	if TX_ChgComp_R.Q and EnaBMSEv01 = TRUE then
		(* BMS_ev21 *)
		EventQueue(EventCode:=81,
			Par1:=DINT_BMS2,
			Par2:=0,
			Par3:=0,
			Par4:=0);
		a:=TRACE_DINT('EventCode', EventQueue.EventCode);
	end_if;

	if TX_ChgComp_R.Q and EnaBMSEv02 = TRUE then
		(* BMS_ev22 *)
		EventQueue(EventCode:=82,
			Par1:=DINT_BMS3,
			Par2:=0,
			Par3:=0,
			Par4:=0);
		a:=TRACE_DINT('EventCode', EventQueue.EventCode);
	end_if;

	if TX_ChgComp_R.Q and EnaBMSEv03 = TRUE then
		(* BMS_ev23 *)
		EventQueue(EventCode:=83,
			Par1:=DINT_BMS_BatV,
			Par2:=0,
			Par3:=0,
			Par4:=0);
		a:=TRACE_DINT('EventCode', EventQueue.EventCode);
	end_if;

	if TX_ChgComp_R.Q and EnaBMSEv04 = TRUE then
		(* BMS_ev24 *)
		EventQueue(EventCode:=84,
			Par1:=DINT_BMS_BatT,
			Par2:=0,
			Par3:=0,
			Par4:=0);
		a:=TRACE_DINT('EventCode', EventQueue.EventCode);
	end_if;

	if TX_ChgComp_R.Q and EnaBMSEv05 = TRUE then
		(* BMS_ev25 *)
		EventQueue(EventCode:=85,
			Par1:=DINT_BMS_BatC,
			Par2:=0,
			Par3:=0,
			Par4:=0);
		a:=TRACE_DINT('EventCode', EventQueue.EventCode);
	end_if;

	if TX_ChgComp_R.Q and EnaBMSEv06 = TRUE then
		(* BMS_ev26 *)
		EventQueue(EventCode:=86,
			Par1:=DINT_BMS_BatA,
			Par2:=0,
			Par3:=0,
			Par4:=0);
		a:=TRACE_DINT('EventCode', EventQueue.EventCode);
	end_if;

	if TX_ChgComp_R.Q and EnaBMSEv07 = TRUE then
		(* BMS_ev27 *)
		EventQueue(EventCode:=87,
			Par1:=DINT_BMS_Main,
			Par2:=0,
			Par3:=0,
			Par4:=0);
		a:=TRACE_DINT('EventCode', EventQueue.EventCode);
	end_if;

	if TX_ChgComp_R.Q and EnaBMSEv08 = TRUE then
		(* BMS_ev28 *)
		EventQueue(EventCode:=88,
			Par1:=DINT_BMS_Chan,
			Par2:=0,
			Par3:=0,
			Par4:=0);
		a:=TRACE_DINT('EventCode', EventQueue.EventCode);
	end_if;

(* Chg_Strt Event*)
	if Chrg_Right_Left_R.Q and EnaBMSEv01 = TRUE then
		(* BMS_ev31 *)
		EventQueue(EventCode:=81,
			Par1:=DINT_BMS2,
			Par2:=0,
			Par3:=0,
			Par4:=0);
		a:=TRACE_DINT('EventCode', EventQueue.EventCode);
	end_if;

	if Chrg_Right_Left_R.Q and EnaBMSEv02 = TRUE then
		(* BMS_ev32 *)
		EventQueue(EventCode:=82,
			Par1:=DINT_BMS3,
			Par2:=0,
			Par3:=0,
			Par4:=0);
		a:=TRACE_DINT('EventCode', EventQueue.EventCode);
	end_if;

	if Chrg_Right_Left_R.Q and EnaBMSEv03 = TRUE then
		(* BMS_ev33 *)
		EventQueue(EventCode:=83,
			Par1:=DINT_BMS_BatV,
			Par2:=0,
			Par3:=0,
			Par4:=0);
		a:=TRACE_DINT('EventCode', EventQueue.EventCode);
	end_if;

	if Chrg_Right_Left_R.Q and EnaBMSEv04 = TRUE then
		(* BMS_ev34 *)
		EventQueue(EventCode:=84,
			Par1:=DINT_BMS_BatT,
			Par2:=0,
			Par3:=0,
			Par4:=0);
		a:=TRACE_DINT('EventCode', EventQueue.EventCode);
	end_if;

	if Chrg_Right_Left_R.Q and EnaBMSEv05 = TRUE then
		(* BMS_ev35 *)
		EventQueue(EventCode:=85,
			Par1:=DINT_BMS_BatC,
			Par2:=0,
			Par3:=0,
			Par4:=0);
		a:=TRACE_DINT('EventCode', EventQueue.EventCode);
	end_if;

	if Chrg_Right_Left_R.Q and EnaBMSEv06 = TRUE then
		(* BMS_ev36 *)
		EventQueue(EventCode:=86,
			Par1:=DINT_BMS_BatA,
			Par2:=0,
			Par3:=0,
			Par4:=0);
		a:=TRACE_DINT('EventCode', EventQueue.EventCode);
	end_if;

	if Chrg_Right_Left_R.Q and EnaBMSEv07 = TRUE then
		(* BMS_ev37 *)
		EventQueue(EventCode:=87,
			Par1:=DINT_BMS_Main,
			Par2:=0,
			Par3:=0,
			Par4:=0);
		a:=TRACE_DINT('EventCode', EventQueue.EventCode);
	end_if;

	if Chrg_Right_Left_R.Q and EnaBMSEv08 = TRUE then
		(* BMS_ev38 *)
		EventQueue(EventCode:=88,
			Par1:=DINT_BMS_Chan,
			Par2:=0,
			Par3:=0,
			Par4:=0);
		a:=TRACE_DINT('EventCode', EventQueue.EventCode);
	end_if;

	if Chrg_Right_Left_R.Q and EnaBMSEv09 = TRUE then
		(* BMS_ev39 *)
		EventQueue(EventCode:=89,
			Par1:=DINT_BMS_ID4L,
			Par2:=0,
			Par3:=0,
			Par4:=0);
		a:=TRACE_DINT('EventCode', EventQueue.EventCode);
	end_if;

	if Chrg_Right_Left_R.Q and EnaBMSEv10 = TRUE then
		(* BMS_ev40 *)
		EventQueue(EventCode:=90,
			Par1:=DINT_BMS_ID4H,
			Par2:=0,
			Par3:=0,
			Par4:=0);
		a:=TRACE_DINT('EventCode', EventQueue.EventCode);
	end_if;

(* Load Event *)
	if TX_Load_R.Q and EnaBMSEv01 = TRUE then
		(* BMS_ev41 *)
		EventQueue(EventCode:=81,
			Par1:=DINT_BMS2,
			Par2:=0,
			Par3:=0,
			Par4:=0);
		a:=TRACE_DINT('EventCode', EventQueue.EventCode);
	end_if;

	if TX_Load_R.Q and EnaBMSEv02 = TRUE then
		(* BMS_ev42 *)
		EventQueue(EventCode:=82,
			Par1:=DINT_BMS3,
			Par2:=0,
			Par3:=0,
			Par4:=0);
		a:=TRACE_DINT('EventCode', EventQueue.EventCode);
	end_if;

	if TX_Load_R.Q and EnaBMSEv03 = TRUE then
		(* BMS_ev43 *)
		EventQueue(EventCode:=83,
			Par1:=DINT_BMS_BatV,
			Par2:=0,
			Par3:=0,
			Par4:=0);
		a:=TRACE_DINT('EventCode', EventQueue.EventCode);
	end_if;

	if TX_Load_R.Q and EnaBMSEv04 = TRUE then
		(* BMS_ev44 *)
		EventQueue(EventCode:=84,
			Par1:=DINT_BMS_BatT,
			Par2:=0,
			Par3:=0,
			Par4:=0);
		a:=TRACE_DINT('EventCode', EventQueue.EventCode);
	end_if;

	if TX_Load_R.Q and EnaBMSEv05 = TRUE then
		(* BMS_ev45 *)
		EventQueue(EventCode:=85,
			Par1:=DINT_BMS_BatC,
			Par2:=0,
			Par3:=0,
			Par4:=0);
		a:=TRACE_DINT('EventCode', EventQueue.EventCode);
	end_if;

	if TX_Load_R.Q and EnaBMSEv06 = TRUE then
		(* BMS_ev46 *)
		EventQueue(EventCode:=86,
			Par1:=DINT_BMS_BatA,
			Par2:=0,
			Par3:=0,
			Par4:=0);
		a:=TRACE_DINT('EventCode', EventQueue.EventCode);
	end_if;

	if TX_Load_R.Q and EnaBMSEv07 = TRUE then
		(* BMS_ev47 *)
		EventQueue(EventCode:=87,
			Par1:=DINT_BMS_Main,
			Par2:=0,
			Par3:=0,
			Par4:=0);
		a:=TRACE_DINT('EventCode', EventQueue.EventCode);
	end_if;

	if TX_Load_R.Q and EnaBMSEv08 = TRUE then
		(* BMS_ev48 *)
		EventQueue(EventCode:=88,
			Par1:=DINT_BMS_Chan,
			Par2:=0,
			Par3:=0,
			Par4:=0);
		a:=TRACE_DINT('EventCode', EventQueue.EventCode);
	end_if;

(* Error event *)

NDC8.OMPLC.ChargeOM := WORD_TO_INT(OM_PLC_Word1);
NDC8.OMPLC.Stop_OM := WORD_TO_INT(OM_PLC_Word2);

END_FUNCTION_BLOCK
